// TIA Portal V16 export
// export: Created 2023-09-11T12:14:52.9400117Z, ExportSetting WithDefaults, DisplayName Totally Integrated Automation Portal, DisplayVersion V16 Update 6, DisplayName TIA Portal Version Control Interface, DisplayVersion V16 Update 2, DisplayName TIA Portal Openness, DisplayVersion V16 Update 6, DisplayName STEP 7 Professional, DisplayVersion V16 Update 6, DisplayName STEP 7 Safety, DisplayVersion V16, DisplayName WinCC Advanced, DisplayVersion V16 Update 6
FUNCTION_BLOCK "06_M_Control strategy Pumping station"   // FB4, LAD
TITLE = Ustawienie metody sterowania
{ S7_Optimized_Access := 'TRUE' }
AUTHOR : rtecmer
VERSION : 0.1
// stored: AutoNumber true, IsIECCheckEnabled false, IsRetainMemResEnabled false, MemoryReserve 100, SetENOAutomatically false, UDAEnableTagReadback false
   VAR_INPUT
      tempStrategia_Pompownia : Int;   // Słowo strategii przechwyconej w FB24
      "bit_alarm_magistrala _min" : Bool;   // bit alarmu niskie ciśniei na magistrali
      bit_off_alarm_magistrala_niskie : Bool;   // bit wyłaczenia alarmu magistrali niskie
   END_VAR
   VAR_IN_OUT
      "Strategia Pompownia" : Int;
   END_VAR
   VAR
      tmp_on_alarm { ExternalAccessible := 'False'; ExternalVisible := 'False'; ExternalWritable := 'False'} : Bool;
      tmp_off_alarm { ExternalAccessible := 'False'; ExternalVisible := 'False'; ExternalWritable := 'False'} : Bool;
      memTriger_set_Strategia { ExternalAccessible := 'False'; ExternalVisible := 'False'; ExternalWritable := 'False'} : Bool;
      memTriger_reset_Strategia { ExternalAccessible := 'False'; ExternalVisible := 'False'; ExternalWritable := 'False'} : Bool;
      test { ExternalAccessible := 'False'; ExternalVisible := 'False'; ExternalWritable := 'False'} : Bool;
   END_VAR
   VAR CONSTANT
      "strategia awaria" : Int := 0;   // regulator wyłączony gdy brak wody w zbiornikach i małae ciśnienie na magistrali
   END_VAR
   VAR_TEMP   // added for the SCL form of the ladder/FBD networks
      _w1 : Bool;
      _w2 : Bool;
   END_VAR
BEGIN

REGION Network 1: Koniec awarii magistrali
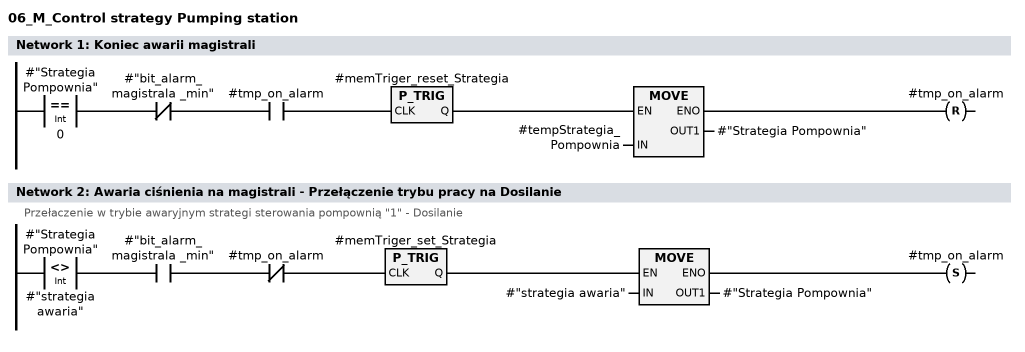
   RUNG wire#powerrail
      { S7_Templates := "SrcType := Int" } EQ_Contact(in1 := #"Strategia Pompownia", in2 := 0)
      I_Contact( #"bit_alarm_magistrala _min" )
      Contact( #tmp_on_alarm )
      P_Trig( #memTriger_reset_Strategia )
      Move(in := #tempStrategia_Pompownia, out1 => #"Strategia Pompownia")
      R_Coil( #tmp_on_alarm )
   END_RUNG
   // the same network as SCL:
   #_w1 := (#"Strategia Pompownia" = 0) AND NOT #"bit_alarm_magistrala _min" AND #tmp_on_alarm;
   #_w2 := #_w1 AND NOT #memTriger_reset_Strategia;   // rising edge
   #memTriger_reset_Strategia := #_w1;
   IF #_w2 THEN
       #"Strategia Pompownia" := #tempStrategia_Pompownia;
       #tmp_on_alarm := FALSE;
   END_IF;
END_REGION

REGION Network 2: Awaria ciśnienia na magistrali - Przełączenie trybu pracy na Dosilanie
   // Przełaczenie w trybie awaryjnym strategi sterowania pompownią "1" - Dosilanie
   RUNG wire#powerrail
      { S7_Templates := "SrcType := Int" } NE_Contact(in1 := #"Strategia Pompownia", in2 := #"strategia awaria")
      Contact( #"bit_alarm_magistrala _min" )
      I_Contact( #tmp_on_alarm )
      P_Trig( #memTriger_set_Strategia )
      Move(in := #"strategia awaria", out1 => #"Strategia Pompownia")
      S_Coil( #tmp_on_alarm )
   END_RUNG
   // the same network as SCL:
   #_w1 := (#"Strategia Pompownia" <> #"strategia awaria") AND #"bit_alarm_magistrala _min" AND NOT #tmp_on_alarm;
   #_w2 := #_w1 AND NOT #memTriger_set_Strategia;   // rising edge
   #memTriger_set_Strategia := #_w1;
   IF #_w2 THEN
       #"Strategia Pompownia" := #"strategia awaria";
       #tmp_on_alarm := TRUE;
   END_IF;
END_REGION
END_FUNCTION_BLOCK
